Staubli VAL3: flagStatus.pjx

Parameters version=s7.9.1 stackSize=5000 millimeterUnit=true
Data file=flagStatus.dtx
